Fanuc KAREL source: NC0048.KL

-- PROVISIONAL review KL for V1013-1; original PC SHA256 0264e25870972dbb108cd1eb54df17dc74f507463d0907c5a15b50d9dce7201e
-- Incomplete behavior may be omitted. Consult companion uncertainty JSON. Do not deploy.
PROGRAM NC0048
%NOLOCKGROUP
-- UNRESOLVED_LOCAL_POOL 1 cells at code offset 3; source declarations unknown
-- DIRECT_LOCAL_WORD_ACCESS alone does not prove INTEGER, REAL, or BOOLEAN
BEGIN
  -- UNRESOLVED_PC offsets 0-8; opcodes 2B,2C,7B
  -- UNRESOLVED_PC offsets 13-20; opcodes 9D,23
  -- UNRESOLVED_PC offsets 25-38; opcodes 21,9D,57,79
  -- UNRESOLVED_PC offsets 43-60; opcodes 21,40,41,42
  -- UNRESOLVED_PC offsets 65-78; opcodes 21,9D,57,79
  -- UNRESOLVED_PC offsets 83-100; opcodes 21,40,41,42
  -- UNRESOLVED_PC offsets 105-118; opcodes 21,9D,57,79
  -- UNRESOLVED_PC offsets 123-140; opcodes 21,40,41,42
  -- UNRESOLVED_PC offsets 145-158; opcodes 21,9D,57,79
  -- UNRESOLVED_PC offsets 163-180; opcodes 21,40,41,42
  -- UNRESOLVED_PC offsets 185-198; opcodes 21,9D,57,79
  -- UNRESOLVED_PC offsets 203-220; opcodes 21,40,41,42
  -- UNRESOLVED_PC offsets 225-238; opcodes 21,9D,57,79
  -- UNRESOLVED_PC offsets 243-260; opcodes 21,40,41,42
  -- UNRESOLVED_PC offsets 265-295; opcodes 21,9D,52,23,7A,40,41,42
  -- UNRESOLVED_PC offsets 300-324; opcodes 21,2E,52,23,7A,43
  -- UNRESOLVED_PC offsets 329-347; opcodes 21,2E,52,23
  -- UNRESOLVED_PC offsets 357-362; opcodes 7A
  -- UNRESOLVED_PC offsets 367-385; opcodes 21,2E,52,23
  -- UNRESOLVED_PC offsets 390-406; opcodes 7A,40,41,42
  -- UNRESOLVED_PC offsets 411-435; opcodes 21,2E,52,23,7A,43
  -- UNRESOLVED_PC offsets 440-458; opcodes 21,2E,52,23
  -- UNRESOLVED_PC offsets 468-473; opcodes 7A
  -- UNRESOLVED_PC offsets 478-496; opcodes 21,2E,52,23
  -- UNRESOLVED_PC offsets 501-517; opcodes 7A,40,41,42
  -- UNRESOLVED_PC offsets 522-546; opcodes 21,2E,52,23,7A,43
  -- UNRESOLVED_PC offsets 551-569; opcodes 21,2E,52,23
  -- UNRESOLVED_PC offsets 579-584; opcodes 7A
  -- UNRESOLVED_PC offsets 589-607; opcodes 21,2E,52,23
  -- UNRESOLVED_PC offsets 612-628; opcodes 7A,40,41,42
  -- UNRESOLVED_PC offsets 633-657; opcodes 21,2E,52,23,7A,43
  -- UNRESOLVED_PC offsets 662-680; opcodes 21,2E,52,23
  -- UNRESOLVED_PC offsets 690-695; opcodes 7A
  -- UNRESOLVED_PC offsets 700-718; opcodes 21,2E,52,23
  -- UNRESOLVED_PC offsets 723-739; opcodes 7A,40,41,42
  -- UNRESOLVED_PC offsets 744-768; opcodes 21,2E,52,23,7A,43
  -- UNRESOLVED_PC offsets 773-791; opcodes 21,2E,52,23
  -- UNRESOLVED_PC offsets 801-806; opcodes 7A
  -- UNRESOLVED_PC offsets 811-829; opcodes 21,2E,52,23
  -- UNRESOLVED_PC offsets 834-850; opcodes 7A,40,41,42
  -- UNRESOLVED_PC offsets 855-879; opcodes 21,2E,52,23,7A,43
  -- UNRESOLVED_PC offsets 884-902; opcodes 21,2E,52,23
  -- UNRESOLVED_PC offsets 912-917; opcodes 7A
  -- UNRESOLVED_PC offsets 922-940; opcodes 21,2E,52,23
  -- UNRESOLVED_PC offsets 950-954; opcodes 7F
  -- UNRESOLVED_PC offsets 959-963; opcodes 27,AA
  -- UNRESOLVED_PC offsets 968-972; opcodes 7F
END NC0048
